// TwinCAT 3 PLC project PLC
// Title: SimpleUnitTestExampleProject
// Company: Red Rock Controls Limited
// Author: Roger Christopher
// ProjectVersion: 1.0.4.0
// Description: Updated to use tcl_SimpleUnitTestLibrary V1.0.10.0 tcl_BaseClasses V 1.0.15.0
// ProgramVersion: 3.1.4023.0
// libraries:
//   Tc2_Standard, * (Beckhoff Automation GmbH)
//   Tc2_System, * (Beckhoff Automation GmbH)
//   Tc3_Module, * (Beckhoff Automation GmbH)
//   tcl_BaseClasses, * (Red Rock Controls Limited)
//   tcl_SimpleUnitTestLibrary, * (Red Rock Controls Limited)
// project tree:
//   / GlobalTextList.TcGTLO, PlcTask.TcTTO, Visualization Manager.TcVMO (not stored)
//   POUs/ MAIN.TcPOU
//   POUs/Unit Tests/ PB_TestRunner.TcPOU, Test_FB_Counter_Increments.TcPOU, Test_FB_Counter_SetsQ_Output.TcPOU
//   Version/ Global_Version.TcGVL
//   Visualisation/ Visualization.TcVIS
// real-time tasks:
//   TASK PlcTask: cycle T#10ms, priority 20, ADS port 350

CONFIGURATION PLC
    RESOURCE PLC ON TwinCAT3
        TASK PlcTask(INTERVAL := T#10ms, PRIORITY := 20);
        PROGRAM MAIN WITH PlcTask : MAIN;
    END_RESOURCE
END_CONFIGURATION

// ---- Version/Global_Version.TcGVL
{attribute 'TcGenerated'}
{attribute 'no-analysis'}
{attribute 'linkalways'}
// This function has been automatically generated from the project information.
VAR_GLOBAL CONSTANT
	{attribute 'const_non_replaced'}
	stLibVersion_SimpleUnitTestExampleProject : ST_LibVersion := (iMajor := 1, iMinor := 0, iBuild := 4, iRevision := 0, nFlags := 0, sVersion := '1.0.4.0');
END_VAR

// ---- POUs/MAIN.TcPOU
PROGRAM MAIN
VAR
END_VAR

PB_TestRunner();

END_PROGRAM

// ---- POUs/Unit Tests/PB_TestRunner.TcPOU
PROGRAM PB_TestRunner
VAR
    TestRunner : T_TestRunner;
    
    // Test Suite holds a list of tests that are automatically added to list of tests held by the test framework...
    FB_Counter_Tests : T_TestSuite;
    Test_FB_Counter_Increments   : Test_FB_Counter_Increments  (TestSuite := FB_Counter_Tests); 
    Test_FB_Counter_SetsQ_Output : Test_FB_Counter_SetsQ_Output(TestSuite := FB_Counter_Tests);
END_VAR

IF TestRunner.ReloadTests THEN
    TestRunner.AddTestSuite(FB_Counter_Tests); // Run tests defined in this project
    TestRunner.ReloadTests := FALSE;
END_IF

TestRunner();

END_PROGRAM

// ---- POUs/Unit Tests/Test_FB_Counter_Increments.TcPOU
FUNCTION_BLOCK Test_FB_Counter_Increments EXTENDS T_UnitTestBase
VAR
    Counter : CTU;
END_VAR

// Setup..
Counter(
	CU:= FALSE, 
	RESET:= TRUE, 
	PV:= , 
	Q=> , 
	CV=> );

// Test... 
Counter(
	CU:= TRUE, 
	RESET:= FALSE, 
	PV:= , 
	Q=> , 
	CV=> );
// Verify...   
Assertion.AssertEquals_WORD(
    Expected:= 1, 
    Actual:= Counter.CV, 
    VariableName:= 'Counter.CV');   

// Done...   
TestFinished();

END_FUNCTION_BLOCK

// ---- POUs/Unit Tests/Test_FB_Counter_SetsQ_Output.TcPOU
FUNCTION_BLOCK Test_FB_Counter_SetsQ_Output EXTENDS T_UnitTestBase
VAR
    Counter : CTU;
END_VAR

// Setup..
Counter(
	CU:= FALSE, 
	RESET:= TRUE, 
	PV:= 1, 
	Q=> , 
	CV=> );

// Test... 
Counter(
	CU:= TRUE, 
	RESET:= FALSE, 
	PV:= , 
	Q=> , 
	CV=> );
// Verify...   
Assertion.AssertEquals_BOOL(
    Expected:= TRUE, 
    Actual:= Counter.Q, 
    VariableName:= 'Counter.Q');   

// Done...   
TestFinished();

END_FUNCTION_BLOCK

// ---- Visualisation/Visualization.TcVIS
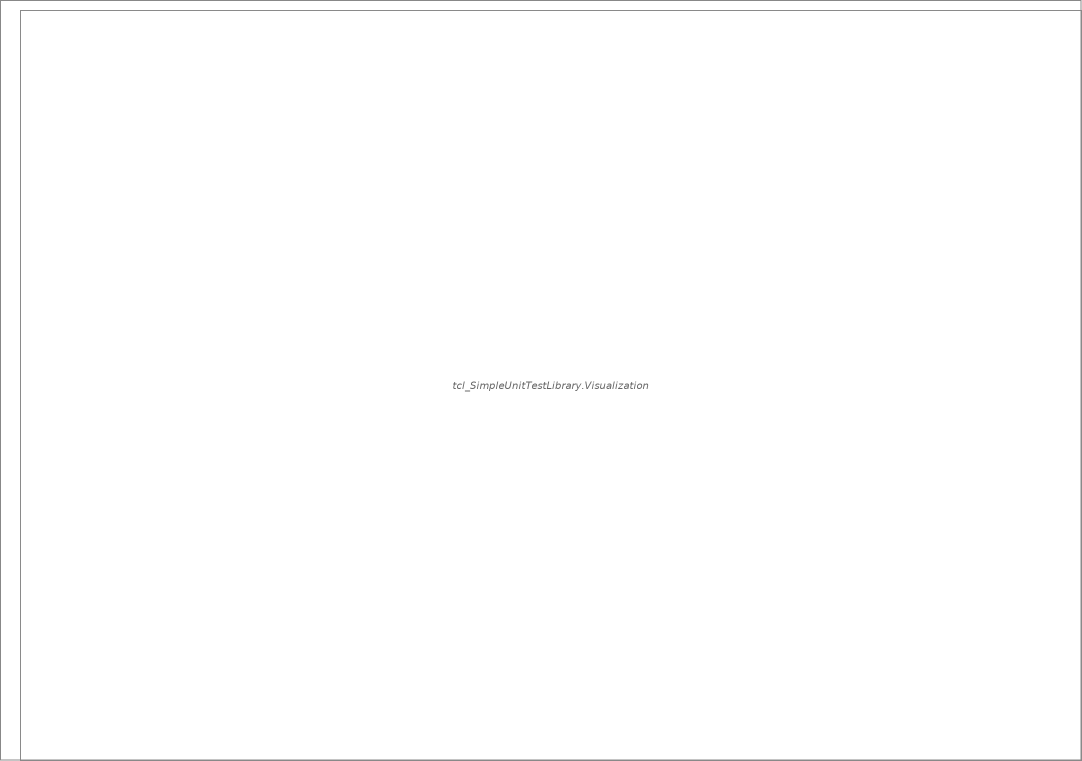
VISUALIZATION Visualization  // 1082x761
    Frame (20,10 1062x751)
        shows tcl_SimpleUnitTestLibrary.Visualization(TestRunner := PB_TestRunner.TestRunner)
END_VISUALIZATION
